// TIA Portal V17 export
// export: Created 2026-04-13T11:12:44.5384284Z, ExportSetting WithDefaults, DisplayName Totally Integrated Automation Portal, DisplayVersion V17 Update 4, DisplayName TIA Portal Openness, DisplayVersion V17 Update 4, DisplayName TIA Portal Version Control Interface, DisplayVersion V17, DisplayName SINAMICS Startdrive Advanced, DisplayVersion V17, DisplayName SINAMICS Startdrive G130, G150, S120, S150, SINAMICS MV, S210, DisplayVersion V17, DisplayName SINAMICS Startdrive G110M, G120, G120C, G120D, G120P, G115D, DisplayVersion V17, DisplayName STEP 7 Professional, DisplayVersion V17 Update 4, DisplayName STEP 7 Safety, DisplayVersion V17, DisplayName WinCC Professional, DisplayVersion V17 Update 4
DATA_BLOCK "C2-闭式自动_DB"   // DB20
VERSION : 0.1
// stored: AutoNumber true, DBAccessibleFromOPCUA true, DBAccessibleFromWebserver true, InstanceOfName C2-闭式自动, InstanceOfType FB
"C2-闭式自动"
   // VAR
   //    闭式自动喷雾 { S7_SetPoint := 'True'} : "闭式自动喷雾块";
   //    雾化塔保压 { S7_SetPoint := 'True'} : "闭式保压块";
   //    TON1 { S7_SetPoint := 'True'} : TON_TIME;
   //    TON2 { S7_SetPoint := 'True'} : TON_TIME;
   //    TON3 { S7_SetPoint := 'True'} : TON_TIME;
   //    BD布袋反吹记录 { S7_SetPoint := 'True'} : "D3-布袋记录";
   //    FT1 { S7_SetPoint := 'True'} : F_TRIG;
   //    RT1 { S7_SetPoint := 'True'} : R_TRIG;
   //    RT2 { S7_SetPoint := 'True'} : R_TRIG;
   //    TP1 { S7_SetPoint := 'True'} : TP_TIME;
   // END_VAR
BEGIN
END_DATA_BLOCK
